FUNCTION_BLOCK Ass_UnloadNG IMPLEMENTS ITF_AutoStructCommand
VAR_INPUT
END_VAR
VAR_OUTPUT
	SamplingWeight	:REAL;
END_VAR
VAR
	strText,strNGText,strShackText 	:STRING;
	i	:INT;
	_bProcessScan,_bInitialScan: BOOL;
	_bHalt , _bError,_bHaltPause: BOOL;
	nStep,nInitiStep ,nNGStep,nShackStep 	: INT;
	_tmrT0,tmrLoadcell,tmrshock	,tmrNG		:TON;
	bBoxPass: BOOL;
	tmrClear: TON;
	UpperWeight,LowerWeight	:REAL;
END_VAR

IF NOT _bInitialScan AND NOT _bProcessScan THEN
	strText:=strNGText:=strShackText	:='';
END_IF


IF NOT _bInitialScan THEN
	nInitiStep	:= 0;
END_IF

_bInitialScan:=FALSE;



IF NOT _bProcessScan THEN
	nShackStep	:= 0;
	nNGStep		:= 0;
	nStep		:= 0;
END_IF

_bProcessScan	:=FALSE;

{warning 'add property implementation'}
PROPERTY Connect : STRING(50)
GET
END_GET
SET
END_SET
END_PROPERTY

PROPERTY Error : BOOL
GET
END_GET
END_PROPERTY

METHOD ErrorClear : BOOL
_bError	:= FALSE;
END_METHOD

{warning 'add method implementation '}
METHOD FB_init : BOOL
VAR_INPUT
	(* if TRUE, the retain variables are initialized (warm start / cold start)*)
	bInitRetains	: BOOL;
	(* if TRUE, the instance afterwards gets moved into the copy code (online change)*)
	bInCopyCode	: BOOL;
END_VAR
END_METHOD

METHOD HaltStepContiune : BOOL
HaltStepContiune	:=TRUE;
END_METHOD

METHOD Initialization : BOOL
VAR_INPUT
	_Testmode	: BOOL;
END_VAR

VAR
	bConfig: BOOL;
END_VAR
(*
_tmrT0(IN:=TRUE,PT:=T#0.2S);
LoadCell.i_bCmd_Tara:= NOT _tmrT0.Q  ;
Initialization	:= AssRoller.Initialization() AND _tmrT0.Q ;
SamplingWeight	:=0;
Cyl_NGPurge.qExtendCoil	:= FALSE;
Roller_Purge.qRun:= FALSE;
Motor_shock.qRun	:= FALSE;
Motor_shock.qSign	:= FALSE;
Cyl_ShockStop.qExtendCoil:= FALSE;
*)

_bInitialScan:=TRUE;

CASE nInitiStep OF
	0:		
		LoadCell.GetTara();
		_tmrT0(IN:=FALSE);
		strText:='ORG : Initial ';
		Cyl_NGPurge.qExtendCoil		:= FALSE;
		Roller_Purge.qRun			:= FALSE;
		Motor_shock.qRun			:= FALSE;
		Motor_shock.qSign			:= FALSE;
		Cyl_ShockStop.qExtendCoil	:= FALSE;		
		nInitiStep						:= 5;
	5:
		bConfig			:=TRUE;
		IF Sen_TFLoadIn THEN
			bConfig			:=FALSE;
			EventLogger.eEventType		:= 3;
			EventLogger.strEventText	:= 'TF Sensor Error ';	
			EventLogger();					
		END_IF		
			
		IF bConfig THEN
			nInitiStep	:= 10;
			strText:='ORG : Runing ';
			ELSE
			strText:='ORG : Failed ';
			nInitiStep	:= 50;
		END_IF	
	10:
		IF AssRoller.Initialization() THEN
			strText		:='ORG : Done ';
			nInitiStep	:= 20;
		END_IF;		
	20:
		Initialization	:= TRUE;
	
END_CASE;
END_METHOD

{warning 'add property implementation'}
PROPERTY NoEntry : BOOL
GET
END_GET
END_PROPERTY

{warning 'add method implementation '}
METHOD Pause : BOOL
END_METHOD

METHOD Process : BOOL
VAR_INPUT
	bHlatMode	: BOOL;
END_VAR

VAR
	bStoppedComv: BOOL;
END_VAR
_bProcessScan:= TRUE;
//判斷 

CASE nStep OF
	0:
		tmrLoadcell(IN:= FALSE);
		_tmrT0(IN:=FALSE);
		AssRoller.Roller();
		strText:= 'Waiting';
		IF Sen_TFLoadIn THEN
			nStep := 5;
		END_IF
	5:
		strText:= 'Loadind and Stop';
		AssRoller.Roller();
		IF NOT Sen_TFLoadIn THEN
			SamplingWeight	:= 0;
			nStep := 10;
		END_IF	
	10:		
		strText:= 'Weight Check!';
		tmrLoadcell(IN:= TRUE,PT:=T#1S);
		UpperWeight	:= RunParameter.PackagingWeight + RunParameter.PackagingWeightUpLimit ;
		LowerWeight := RunParameter.PackagingWeight - RunParameter.PackagingWeightLowLimit ;
		IF tmrLoadcell.Q THEN
			tmrLoadcell(IN:= FALSE,PT:=T#1S);
			SamplingWeight	:= 	LoadCell.o_rWeight;
			IF SamplingWeight >= LowerWeight AND
				SamplingWeight <= UpperWeight THEN
				strText:= 'Weight Pass!';
				bBoxPass:= TRUE;
				ELSE
				EventLogger.eEventType		:= 2;
				EventLogger.strEventText	:= 'Box Over Weight ';	
				EventLogger.strEventText	:=	CONCAT(EventLogger.strEventText,LEFT(REAL_TO_STRING(SamplingWeight),3));
				EventLogger();
				strText:= 'Box NG';
				bBoxPass:= FALSE;
			END_IF
			nStep := 15;
		END_IF
	
	15:
		
		IF nNGstep = 0 THEN
			nNGstep	:= 5;
			IF RunParameter.PackagingCheck THEN
				bStoppedComv	:= TRUE;
			END_IF
			AssRoller.Belt();
			IF Sen_NGLoadOut THEN
				nStep := 0;
			END_IF;
		END_IF
		
		
		
		
END_CASE;

CASE nNGstep OF
	0:
		strNGText	:= 'Wait BOX';
		tmrNG(IN:=FALSE,PT:=T#2S);
		Roller_Purge.qRun:= TRUE;
		IF Sen_NGLoadOut THEN
			strNGText	:= 'Active Loading';
			nNGstep := 20;
			CASE nStep OF
				0..10:
				strNGText	:= 'Up Loading';
				nNGstep := 50;
			END_CASE
		END_IF
	5:
		strNGText	:= 'TF Loading';
		AssRoller.Belt();
	
		IF Sen_NGLoadOut THEN
			nStep := 0;
			nNGstep	:= 6;
		END_IF
	6:
			IF bBoxPass THEN
				strNGText	:= 'TF LoadIn Stop';
				Roller_Purge.qRun:= FALSE;
				nStep := 0;
				IF nShackStep = 1 THEN
					strNGText	:= 'Go Shack';
					Roller_Purge.qRun:= TRUE;
					nNGstep	:= 10;
				END_IF;
				ELSE
				EventLogger.eEventType		:= 2;
				EventLogger.strEventText	:= 'NG Perge!';		
				EventLogger();		
				strNGText	:= 'TF NG Perge';
				nNGstep	:= 30;
				Roller_Purge.qRun:= FALSE;
			END_IF		

		
	10:
		IF Sen_ShockPos THEN
			strNGText	:= 'Shack ORG';
			nNGstep	:= 0;
		END_IF
	
	
	30://重量Error
		Cyl_NGPurge.qExtendCoil	:= TRUE;
		tmrNG(IN:=TRUE,PT:=T#2S);
		IF tmrNG.Q THEN
			tmrNG(IN:=FALSE);
			nStep := 0;
			Cyl_NGPurge.qExtendCoil	:= FALSE;
			nNGstep := 0;
		END_IF		
		
		
		
	50://手動投入	
		strNGText	:= '50 Man. ';
		IF Sen_ShockPos THEN
			nNGstep	:= 0;
		END_IF	
END_CASE;	
CASE nShackStep OF
	0:
		tmrshock(IN:=FALSE);
		nShackStep	:= 1;
	1:
		strShackText:='Wait Box';
		Cyl_ShockStop.qExtendCoil:= TRUE;
		tmrshock(IN:=Sen_ShockPos , PT:= RunParameter.shock_DelayTime);	
		Motor_shock.qRun	:= TRUE;
		Motor_shock.qSign	:= TRUE;
		IF tmrshock.q THEN
			strShackText:='Loading Box';
			tmrshock(IN:=FALSE);
			nShackStep	:= 5;
		END_IF
	5:
		strShackText:='Shack Box';
		Motor_shock.qSign	:= FALSE;
		tmrshock(IN:= TRUE, PT:= RunParameter.shock_HighTime);
		IF tmrshock.Q THEN
			tmrshock(IN:= FALSE);
			Motor_shock.qSign	:= TRUE;
			Cyl_ShockStop.qExtendCoil:= FALSE;
			nShackStep	:= 10;
		END_IF
	10:
		strShackText:='Load Out Box';
		tmrshock(IN:= NOT Sen_ShockPos , PT:= T#3S);				

		IF tmrshock.Q THEN
			Cyl_ShockStop.qExtendCoil:= TRUE;
			tmrshock(IN:= FALSE);
			nShackStep	:= 0;
		END_IF
		
		
END_CASE;
END_METHOD

PROPERTY Status : STRING(50)
GET
Status:= strText;
END_GET
END_PROPERTY

END_FUNCTION_BLOCK

(* stored: Version 1.1.0.1, ProductVersion 3.1.4024.16
   POU Ass_UnloadNG: Id {bd20b21e-c1a4-4f4a-a1c0-5aa3b9f16856}, SpecialFunc None
   Property Connect: Id {7225ef76-d320-4fde-b0b3-07f6324857c3}
   Get Get: Id {0f06e400-442d-4c8e-8f47-be25bc937442}
   Set Set: Id {57347063-56a4-46db-bfbe-6d877c2c7926}
   Property Error: Id {d7b9b006-e839-4929-8fdc-7010c3300995}
   Get Get: Id {2e11e90e-71a3-468d-a838-7f96fa2308b3}
   Method ErrorClear: Id {9e2dccef-ea8c-4272-a85c-282b842d5368}
   Method FB_init: Id {30c9c290-32c6-4a77-84b3-c0d393f44a22}
   Method HaltStepContiune: Id {0d812bd6-7f5d-43aa-82ad-0ec04ed19982}
   Method Initialization: Id {590597e0-2263-4555-812b-e1b41a0161a3}
   Property NoEntry: Id {6976b88a-7ea7-42c4-925d-1fa73aaa0fbb}
   Get Get: Id {122c4eba-99f8-44e6-94a8-463d6fbe8b8d}
   Method Pause: Id {a877b4d4-c843-4482-9061-6c3f8d9f1f13}
   Method Process: Id {30f199c4-bbb5-40fe-ab57-f5f98610f032}
   Property Status: Id {54765cf9-d21f-45b1-92d3-fce37714c6cc}
   Get Get: Id {f5aa3595-cea0-42a9-bce6-727859e4b572} *)
